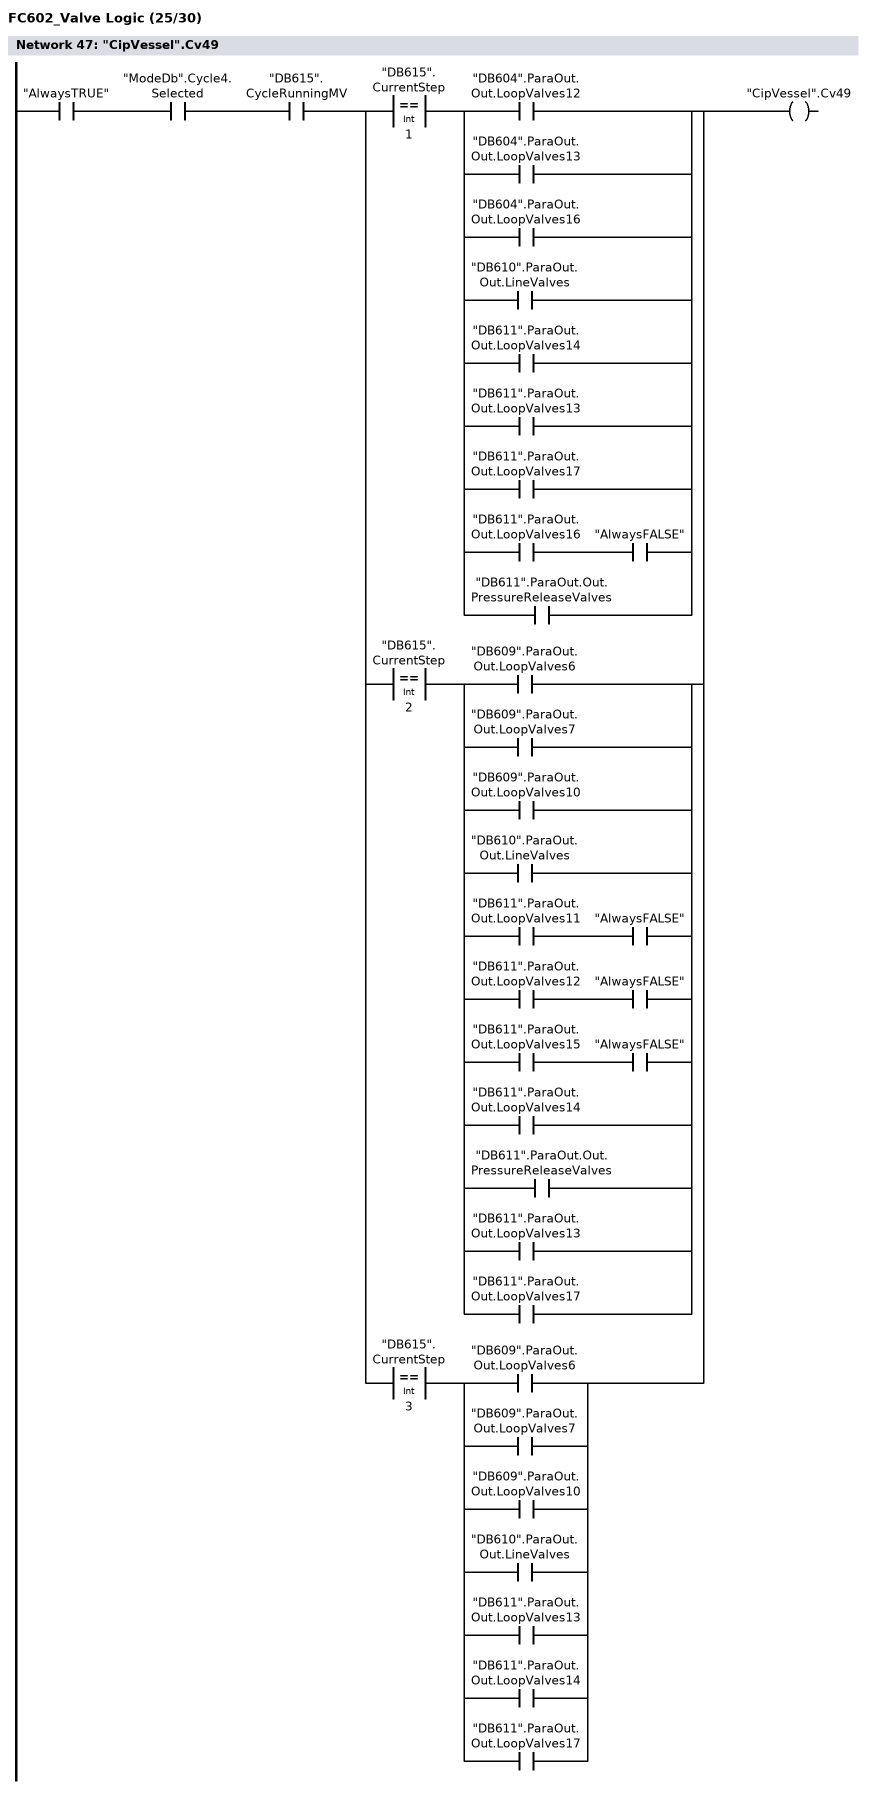
   RUNG wire#powerrail
      Contact( "AlwaysTRUE" )
      Contact( "ModeDb".Cycle4.Selected )
      Contact( "DB615".CycleRunningMV )
      wire#w1
      { S7_Templates := "SrcType := Int" } EQ_Contact(in1 := "DB615".CurrentStep, in2 := 1)
      wire#w2
      Contact( "DB604".ParaOut.Out.LoopValves12 )
      wire#w3
      Coil( "CipVessel".Cv49 )
   END_RUNG
   RUNG wire#w2
      Contact( "DB604".ParaOut.Out.LoopValves13 )
   END_RUNG wire#w3
   RUNG wire#w2
      Contact( "DB604".ParaOut.Out.LoopValves16 )
   END_RUNG wire#w3
   RUNG wire#w2
      Contact( "DB610".ParaOut.Out.LineValves )
   END_RUNG wire#w3
   RUNG wire#w2
      Contact( "DB611".ParaOut.Out.LoopValves14 )
   END_RUNG wire#w3
   RUNG wire#w2
      Contact( "DB611".ParaOut.Out.LoopValves13 )
   END_RUNG wire#w3
   RUNG wire#w2
      Contact( "DB611".ParaOut.Out.LoopValves17 )
   END_RUNG wire#w3
   RUNG wire#w2
      Contact( "DB611".ParaOut.Out.LoopValves16 )
      Contact( "AlwaysFALSE" )
   END_RUNG wire#w3
   RUNG wire#w2
      Contact( "DB611".ParaOut.Out.PressureReleaseValves )
   END_RUNG wire#w3
   RUNG wire#w1
      { S7_Templates := "SrcType := Int" } EQ_Contact(in1 := "DB615".CurrentStep, in2 := 2)
      wire#w4
      Contact( "DB609".ParaOut.Out.LoopValves6 )
   END_RUNG wire#w3
   RUNG wire#w4
      Contact( "DB609".ParaOut.Out.LoopValves7 )
   END_RUNG wire#w3
   RUNG wire#w4
      Contact( "DB609".ParaOut.Out.LoopValves10 )
   END_RUNG wire#w3
   RUNG wire#w4
      Contact( "DB610".ParaOut.Out.LineValves )
   END_RUNG wire#w3
   RUNG wire#w4
      Contact( "DB611".ParaOut.Out.LoopValves11 )
      Contact( "AlwaysFALSE" )
   END_RUNG wire#w3
   RUNG wire#w4
      Contact( "DB611".ParaOut.Out.LoopValves12 )
      Contact( "AlwaysFALSE" )
   END_RUNG wire#w3
   RUNG wire#w4
      Contact( "DB611".ParaOut.Out.LoopValves15 )
      Contact( "AlwaysFALSE" )
   END_RUNG wire#w3
   RUNG wire#w4
      Contact( "DB611".ParaOut.Out.LoopValves14 )
   END_RUNG wire#w3
   RUNG wire#w4
      Contact( "DB611".ParaOut.Out.PressureReleaseValves )
   END_RUNG wire#w3
   RUNG wire#w4
      Contact( "DB611".ParaOut.Out.LoopValves13 )
   END_RUNG wire#w3
   RUNG wire#w4
      Contact( "DB611".ParaOut.Out.LoopValves17 )
   END_RUNG wire#w3
   RUNG wire#w1
      { S7_Templates := "SrcType := Int" } EQ_Contact(in1 := "DB615".CurrentStep, in2 := 3)
      wire#w5
      Contact( "DB609".ParaOut.Out.LoopValves6 )
   END_RUNG wire#w3
   RUNG wire#w5
      Contact( "DB609".ParaOut.Out.LoopValves7 )
   END_RUNG wire#w3
   RUNG wire#w5
      Contact( "DB609".ParaOut.Out.LoopValves10 )
   END_RUNG wire#w3
   RUNG wire#w5
      Contact( "DB610".ParaOut.Out.LineValves )
   END_RUNG wire#w3
   RUNG wire#w5
      Contact( "DB611".ParaOut.Out.LoopValves13 )
   END_RUNG wire#w3
   RUNG wire#w5
      Contact( "DB611".ParaOut.Out.LoopValves14 )
   END_RUNG wire#w3
   RUNG wire#w5
      Contact( "DB611".ParaOut.Out.LoopValves17 )
   END_RUNG wire#w3
   // the same network as SCL:
   "CipVessel".Cv49 := "AlwaysTRUE" AND "ModeDb".Cycle4.Selected AND "DB615".CycleRunningMV AND ((("DB615".CurrentStep = 1) AND ("DB604".ParaOut.Out.LoopValves12 OR "DB604".ParaOut.Out.LoopValves13 OR "DB604".ParaOut.Out.LoopValves16 OR "DB610".ParaOut.Out.LineValves OR "DB611".ParaOut.Out.LoopValves14 OR "DB611".ParaOut.Out.LoopValves13 OR "DB611".ParaOut.Out.LoopValves17 OR ("DB611".ParaOut.Out.LoopValves16 AND "AlwaysFALSE") OR "DB611".ParaOut.Out.PressureReleaseValves)) OR (("DB615".CurrentStep = 2) AND ("DB609".ParaOut.Out.LoopValves6 OR "DB609".ParaOut.Out.LoopValves7 OR "DB609".ParaOut.Out.LoopValves10 OR "DB610".ParaOut.Out.LineValves OR ("DB611".ParaOut.Out.LoopValves11 AND "AlwaysFALSE") OR ("DB611".ParaOut.Out.LoopValves12 AND "AlwaysFALSE") OR ("DB611".ParaOut.Out.LoopValves15 AND "AlwaysFALSE") OR "DB611".ParaOut.Out.LoopValves14 OR "DB611".ParaOut.Out.PressureReleaseValves OR "DB611".ParaOut.Out.LoopValves13 OR "DB611".ParaOut.Out.LoopValves17)) OR (("DB615".CurrentStep = 3) AND ("DB609".ParaOut.Out.LoopValves6 OR "DB609".ParaOut.Out.LoopValves7 OR "DB609".ParaOut.Out.LoopValves10 OR "DB610".ParaOut.Out.LineValves OR "DB611".ParaOut.Out.LoopValves13 OR "DB611".ParaOut.Out.LoopValves14 OR "DB611".ParaOut.Out.LoopValves17)));
END_REGION

REGION Network 48: "CipVessel".Cv53
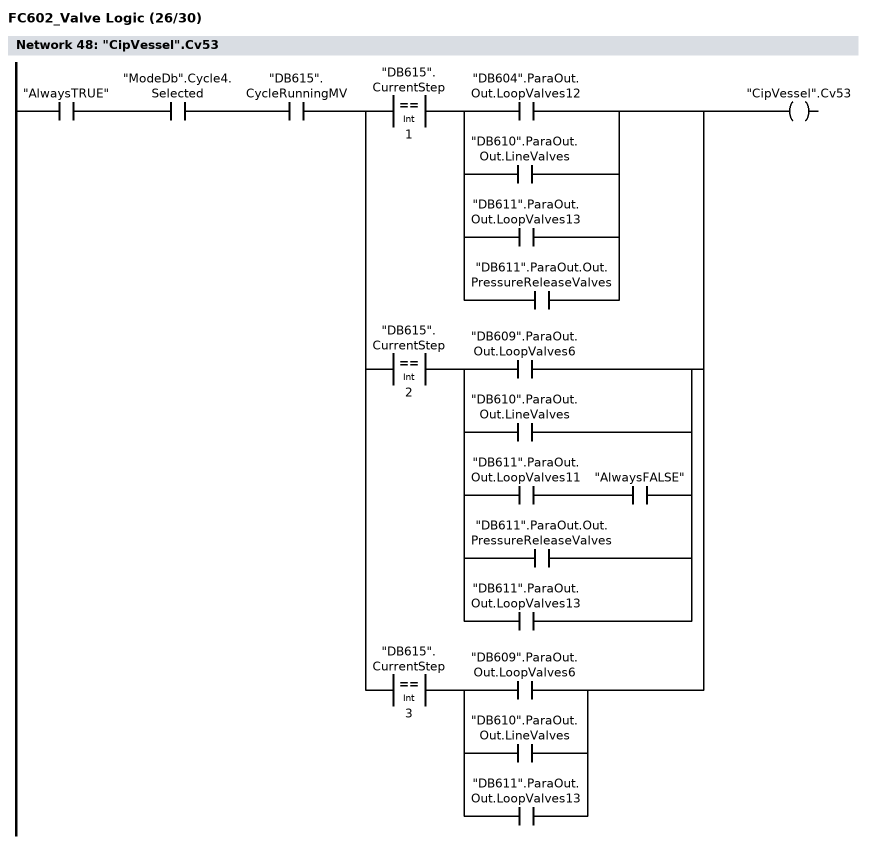
   RUNG wire#powerrail
      Contact( "AlwaysTRUE" )
      Contact( "ModeDb".Cycle4.Selected )
      Contact( "DB615".CycleRunningMV )
      wire#w1
      { S7_Templates := "SrcType := Int" } EQ_Contact(in1 := "DB615".CurrentStep, in2 := 1)
      wire#w2
      Contact( "DB604".ParaOut.Out.LoopValves12 )
      wire#w3
      Coil( "CipVessel".Cv53 )
   END_RUNG
   RUNG wire#w2
      Contact( "DB610".ParaOut.Out.LineValves )
   END_RUNG wire#w3
   RUNG wire#w2
      Contact( "DB611".ParaOut.Out.LoopValves13 )
   END_RUNG wire#w3
   RUNG wire#w2
      Contact( "DB611".ParaOut.Out.PressureReleaseValves )
   END_RUNG wire#w3
   RUNG wire#w1
      { S7_Templates := "SrcType := Int" } EQ_Contact(in1 := "DB615".CurrentStep, in2 := 2)
      wire#w4
      Contact( "DB609".ParaOut.Out.LoopValves6 )
   END_RUNG wire#w3
   RUNG wire#w4
      Contact( "DB610".ParaOut.Out.LineValves )
   END_RUNG wire#w3
   RUNG wire#w4
      Contact( "DB611".ParaOut.Out.LoopValves11 )
      Contact( "AlwaysFALSE" )
   END_RUNG wire#w3
   RUNG wire#w4
      Contact( "DB611".ParaOut.Out.PressureReleaseValves )
   END_RUNG wire#w3
   RUNG wire#w4
      Contact( "DB611".ParaOut.Out.LoopValves13 )
   END_RUNG wire#w3
   RUNG wire#w1
      { S7_Templates := "SrcType := Int" } EQ_Contact(in1 := "DB615".CurrentStep, in2 := 3)
      wire#w5
      Contact( "DB609".ParaOut.Out.LoopValves6 )
   END_RUNG wire#w3
   RUNG wire#w5
      Contact( "DB610".ParaOut.Out.LineValves )
   END_RUNG wire#w3
   RUNG wire#w5
      Contact( "DB611".ParaOut.Out.LoopValves13 )
   END_RUNG wire#w3
   // the same network as SCL:
   "CipVessel".Cv53 := "AlwaysTRUE" AND "ModeDb".Cycle4.Selected AND "DB615".CycleRunningMV AND ((("DB615".CurrentStep = 1) AND ("DB604".ParaOut.Out.LoopValves12 OR "DB610".ParaOut.Out.LineValves OR "DB611".ParaOut.Out.LoopValves13 OR "DB611".ParaOut.Out.PressureReleaseValves)) OR (("DB615".CurrentStep = 2) AND ("DB609".ParaOut.Out.LoopValves6 OR "DB610".ParaOut.Out.LineValves OR ("DB611".ParaOut.Out.LoopValves11 AND "AlwaysFALSE") OR "DB611".ParaOut.Out.PressureReleaseValves OR "DB611".ParaOut.Out.LoopValves13)) OR (("DB615".CurrentStep = 3) AND ("DB609".ParaOut.Out.LoopValves6 OR "DB610".ParaOut.Out.LineValves OR "DB611".ParaOut.Out.LoopValves13)));
END_REGION

REGION Network 49: ----------- PF02 OUT -------------
END_REGION

REGION Network 50: "CipVessel".Cv56
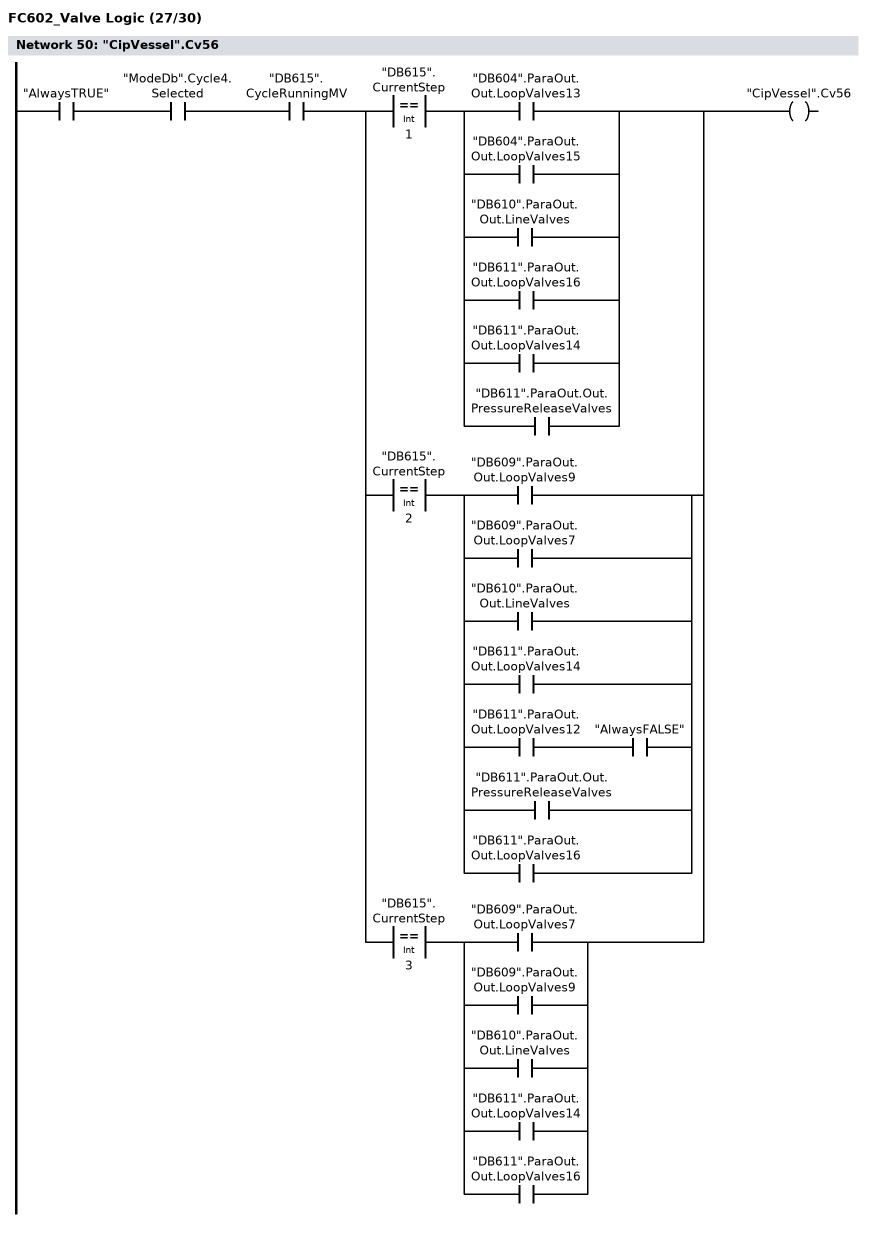
   RUNG wire#powerrail
      Contact( "AlwaysTRUE" )
      Contact( "ModeDb".Cycle4.Selected )
      Contact( "DB615".CycleRunningMV )
      wire#w1
      { S7_Templates := "SrcType := Int" } EQ_Contact(in1 := "DB615".CurrentStep, in2 := 1)
      wire#w2
      Contact( "DB604".ParaOut.Out.LoopValves13 )
      wire#w3
      Coil( "CipVessel".Cv56 )
   END_RUNG
   RUNG wire#w2
      Contact( "DB604".ParaOut.Out.LoopValves15 )
   END_RUNG wire#w3
   RUNG wire#w2
      Contact( "DB610".ParaOut.Out.LineValves )
   END_RUNG wire#w3
   RUNG wire#w2
      Contact( "DB611".ParaOut.Out.LoopValves16 )
   END_RUNG wire#w3
   RUNG wire#w2
      Contact( "DB611".ParaOut.Out.LoopValves14 )
   END_RUNG wire#w3
   RUNG wire#w2
      Contact( "DB611".ParaOut.Out.PressureReleaseValves )
   END_RUNG wire#w3
   RUNG wire#w1
      { S7_Templates := "SrcType := Int" } EQ_Contact(in1 := "DB615".CurrentStep, in2 := 2)
      wire#w4
      Contact( "DB609".ParaOut.Out.LoopValves9 )
   END_RUNG wire#w3
   RUNG wire#w4
      Contact( "DB609".ParaOut.Out.LoopValves7 )
   END_RUNG wire#w3
   RUNG wire#w4
      Contact( "DB610".ParaOut.Out.LineValves )
   END_RUNG wire#w3
   RUNG wire#w4
      Contact( "DB611".ParaOut.Out.LoopValves14 )
   END_RUNG wire#w3
   RUNG wire#w4
      Contact( "DB611".ParaOut.Out.LoopValves12 )
      Contact( "AlwaysFALSE" )
   END_RUNG wire#w3
   RUNG wire#w4
      Contact( "DB611".ParaOut.Out.PressureReleaseValves )
   END_RUNG wire#w3
   RUNG wire#w4
      Contact( "DB611".ParaOut.Out.LoopValves16 )
   END_RUNG wire#w3
   RUNG wire#w1
      { S7_Templates := "SrcType := Int" } EQ_Contact(in1 := "DB615".CurrentStep, in2 := 3)
      wire#w5
      Contact( "DB609".ParaOut.Out.LoopValves7 )
   END_RUNG wire#w3
   RUNG wire#w5
      Contact( "DB609".ParaOut.Out.LoopValves9 )
   END_RUNG wire#w3
   RUNG wire#w5
      Contact( "DB610".ParaOut.Out.LineValves )
   END_RUNG wire#w3
   RUNG wire#w5
      Contact( "DB611".ParaOut.Out.LoopValves14 )
   END_RUNG wire#w3
   RUNG wire#w5
      Contact( "DB611".ParaOut.Out.LoopValves16 )
   END_RUNG wire#w3
   // the same network as SCL:
   "CipVessel".Cv56 := "AlwaysTRUE" AND "ModeDb".Cycle4.Selected AND "DB615".CycleRunningMV AND ((("DB615".CurrentStep = 1) AND ("DB604".ParaOut.Out.LoopValves13 OR "DB604".ParaOut.Out.LoopValves15 OR "DB610".ParaOut.Out.LineValves OR "DB611".ParaOut.Out.LoopValves16 OR "DB611".ParaOut.Out.LoopValves14 OR "DB611".ParaOut.Out.PressureReleaseValves)) OR (("DB615".CurrentStep = 2) AND ("DB609".ParaOut.Out.LoopValves9 OR "DB609".ParaOut.Out.LoopValves7 OR "DB610".ParaOut.Out.LineValves OR "DB611".ParaOut.Out.LoopValves14 OR ("DB611".ParaOut.Out.LoopValves12 AND "AlwaysFALSE") OR "DB611".ParaOut.Out.PressureReleaseValves OR "DB611".ParaOut.Out.LoopValves16)) OR (("DB615".CurrentStep = 3) AND ("DB609".ParaOut.Out.LoopValves7 OR "DB609".ParaOut.Out.LoopValves9 OR "DB610".ParaOut.Out.LineValves OR "DB611".ParaOut.Out.LoopValves14 OR "DB611".ParaOut.Out.LoopValves16)));
END_REGION

REGION Network 51: "CipVessel".Cv57
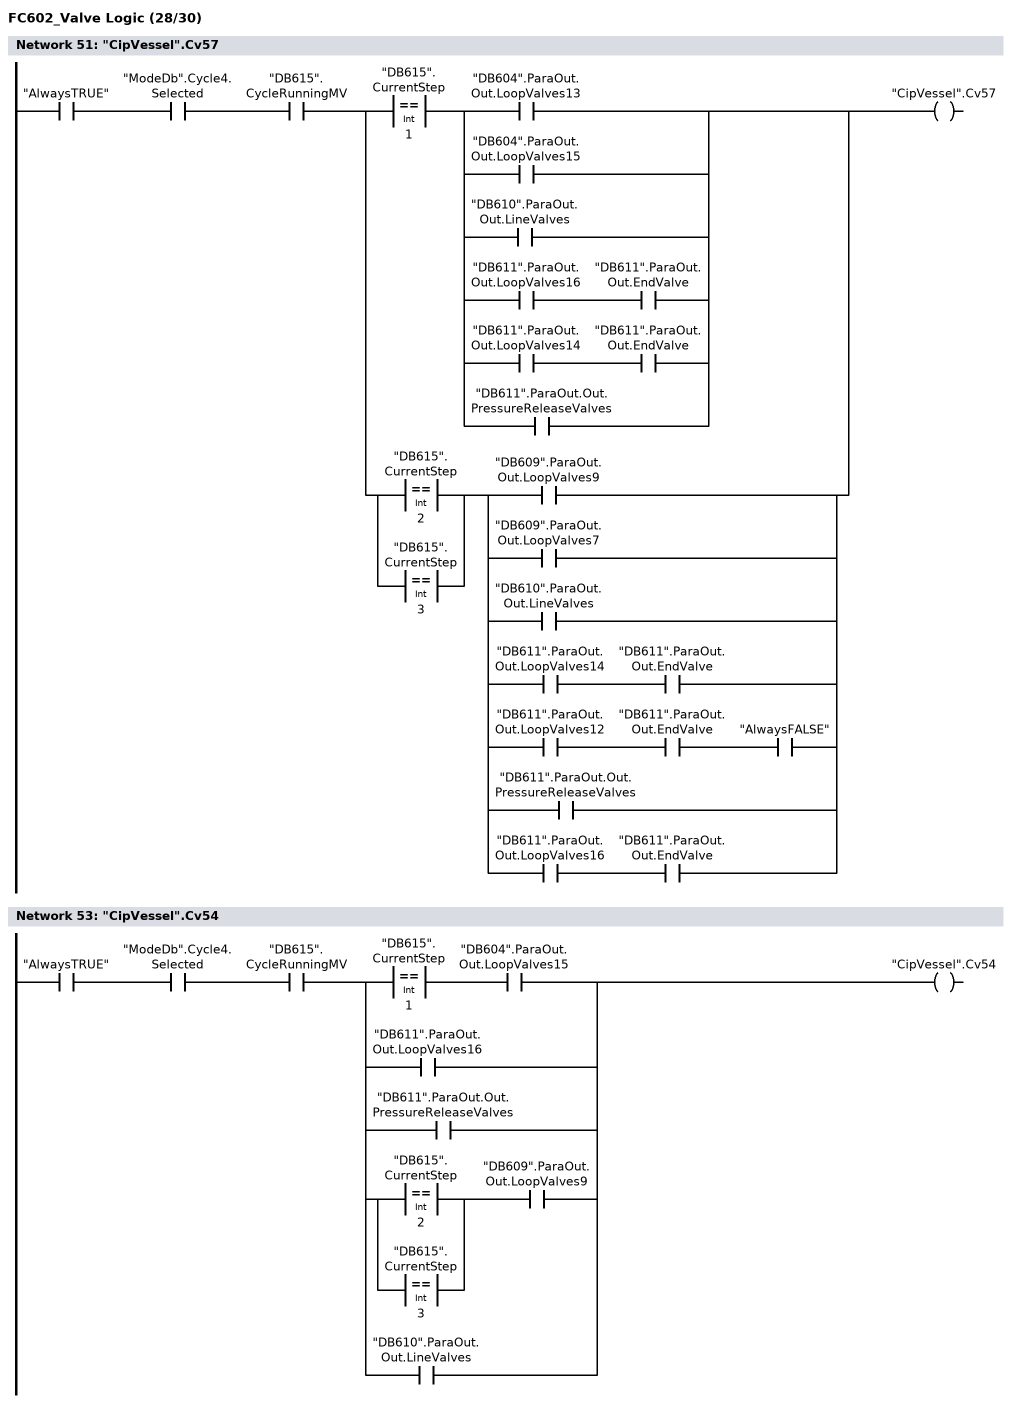
   RUNG wire#powerrail
      Contact( "AlwaysTRUE" )
      Contact( "ModeDb".Cycle4.Selected )
      Contact( "DB615".CycleRunningMV )
      wire#w1
      { S7_Templates := "SrcType := Int" } EQ_Contact(in1 := "DB615".CurrentStep, in2 := 1)
      wire#w2
      Contact( "DB604".ParaOut.Out.LoopValves13 )
      wire#w3
      Coil( "CipVessel".Cv57 )
   END_RUNG
   RUNG wire#w2
      Contact( "DB604".ParaOut.Out.LoopValves15 )
   END_RUNG wire#w3
   RUNG wire#w2
      Contact( "DB610".ParaOut.Out.LineValves )
   END_RUNG wire#w3
   RUNG wire#w2
      Contact( "DB611".ParaOut.Out.LoopValves16 )
      Contact( "DB611".ParaOut.Out.EndValve )
   END_RUNG wire#w3
   RUNG wire#w2
      Contact( "DB611".ParaOut.Out.LoopValves14 )
      Contact( "DB611".ParaOut.Out.EndValve )
   END_RUNG wire#w3
   RUNG wire#w2
      Contact( "DB611".ParaOut.Out.PressureReleaseValves )
   END_RUNG wire#w3
   RUNG wire#w1
      { S7_Templates := "SrcType := Int" } EQ_Contact(in1 := "DB615".CurrentStep, in2 := 2)
      wire#w4
      Contact( "DB609".ParaOut.Out.LoopValves9 )
   END_RUNG wire#w3
   RUNG wire#w1
      { S7_Templates := "SrcType := Int" } EQ_Contact(in1 := "DB615".CurrentStep, in2 := 3)
   END_RUNG wire#w4
   RUNG wire#w4
      Contact( "DB609".ParaOut.Out.LoopValves7 )
   END_RUNG wire#w3
   RUNG wire#w4
      Contact( "DB610".ParaOut.Out.LineValves )
   END_RUNG wire#w3
   RUNG wire#w4
      Contact( "DB611".ParaOut.Out.LoopValves14 )
      Contact( "DB611".ParaOut.Out.EndValve )
   END_RUNG wire#w3
   RUNG wire#w4
      Contact( "DB611".ParaOut.Out.LoopValves12 )
      Contact( "DB611".ParaOut.Out.EndValve )
      Contact( "AlwaysFALSE" )
   END_RUNG wire#w3
   RUNG wire#w4
      Contact( "DB611".ParaOut.Out.PressureReleaseValves )
   END_RUNG wire#w3
   RUNG wire#w4
      Contact( "DB611".ParaOut.Out.LoopValves16 )
      Contact( "DB611".ParaOut.Out.EndValve )
   END_RUNG wire#w3
   // the same network as SCL:
   "CipVessel".Cv57 := "AlwaysTRUE" AND "ModeDb".Cycle4.Selected AND "DB615".CycleRunningMV AND ((("DB615".CurrentStep = 1) AND ("DB604".ParaOut.Out.LoopValves13 OR "DB604".ParaOut.Out.LoopValves15 OR "DB610".ParaOut.Out.LineValves OR ("DB611".ParaOut.Out.LoopValves16 AND "DB611".ParaOut.Out.EndValve) OR ("DB611".ParaOut.Out.LoopValves14 AND "DB611".ParaOut.Out.EndValve) OR "DB611".ParaOut.Out.PressureReleaseValves)) OR ((("DB615".CurrentStep = 2) OR ("DB615".CurrentStep = 3)) AND ("DB609".ParaOut.Out.LoopValves9 OR "DB609".ParaOut.Out.LoopValves7 OR "DB610".ParaOut.Out.LineValves OR ("DB611".ParaOut.Out.LoopValves14 AND "DB611".ParaOut.Out.EndValve) OR ("DB611".ParaOut.Out.LoopValves12 AND "DB611".ParaOut.Out.EndValve AND "AlwaysFALSE") OR "DB611".ParaOut.Out.PressureReleaseValves OR ("DB611".ParaOut.Out.LoopValves16 AND "DB611".ParaOut.Out.EndValve))));
END_REGION

REGION Network 52: ---------- PTL LINE ------------
END_REGION

REGION Network 53: "CipVessel".Cv54
   RUNG wire#powerrail
      Contact( "AlwaysTRUE" )
      Contact( "ModeDb".Cycle4.Selected )
      Contact( "DB615".CycleRunningMV )
      wire#w1
      { S7_Templates := "SrcType := Int" } EQ_Contact(in1 := "DB615".CurrentStep, in2 := 1)
      Contact( "DB604".ParaOut.Out.LoopValves15 )
      wire#w2
      Coil( "CipVessel".Cv54 )
   END_RUNG
   RUNG wire#w1
      Contact( "DB611".ParaOut.Out.LoopValves16 )
   END_RUNG wire#w2
   RUNG wire#w1
      Contact( "DB611".ParaOut.Out.PressureReleaseValves )
   END_RUNG wire#w2
   RUNG wire#w1
      { S7_Templates := "SrcType := Int" } EQ_Contact(in1 := "DB615".CurrentStep, in2 := 2)
      wire#w3
      Contact( "DB609".ParaOut.Out.LoopValves9 )
   END_RUNG wire#w2
   RUNG wire#w1
      { S7_Templates := "SrcType := Int" } EQ_Contact(in1 := "DB615".CurrentStep, in2 := 3)
   END_RUNG wire#w3
   RUNG wire#w1
      Contact( "DB610".ParaOut.Out.LineValves )
   END_RUNG wire#w2
   // the same network as SCL:
   "CipVessel".Cv54 := "AlwaysTRUE" AND "ModeDb".Cycle4.Selected AND "DB615".CycleRunningMV AND ((("DB615".CurrentStep = 1) AND "DB604".ParaOut.Out.LoopValves15) OR "DB611".ParaOut.Out.LoopValves16 OR "DB611".ParaOut.Out.PressureReleaseValves OR ((("DB615".CurrentStep = 2) OR ("DB615".CurrentStep = 3)) AND "DB609".ParaOut.Out.LoopValves9) OR "DB610".ParaOut.Out.LineValves);
END_REGION

REGION Network 54: "CipVessel".Cv55
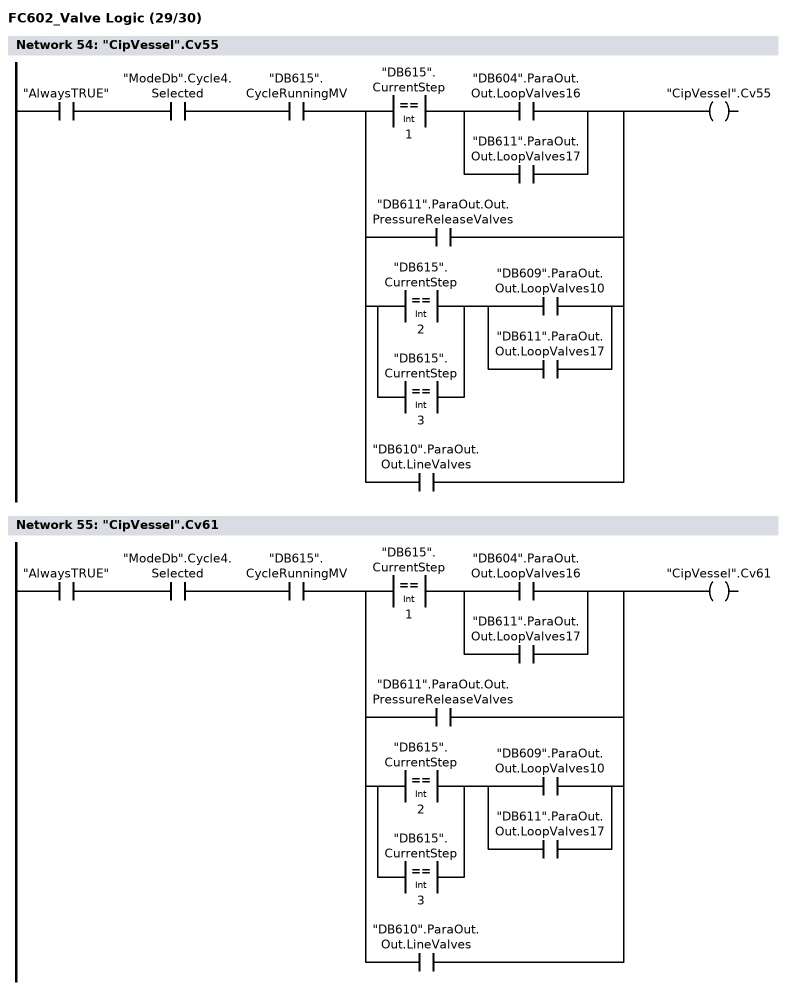
   RUNG wire#powerrail
      Contact( "AlwaysTRUE" )
      Contact( "ModeDb".Cycle4.Selected )
      Contact( "DB615".CycleRunningMV )
      wire#w1
      { S7_Templates := "SrcType := Int" } EQ_Contact(in1 := "DB615".CurrentStep, in2 := 1)
      wire#w2
      Contact( "DB604".ParaOut.Out.LoopValves16 )
      wire#w3
      Coil( "CipVessel".Cv55 )
   END_RUNG
   RUNG wire#w2
      Contact( "DB611".ParaOut.Out.LoopValves17 )
   END_RUNG wire#w3
   RUNG wire#w1
      Contact( "DB611".ParaOut.Out.PressureReleaseValves )
   END_RUNG wire#w3
   RUNG wire#w1
      { S7_Templates := "SrcType := Int" } EQ_Contact(in1 := "DB615".CurrentStep, in2 := 2)
      wire#w4
      Contact( "DB609".ParaOut.Out.LoopValves10 )
   END_RUNG wire#w3
   RUNG wire#w1
      { S7_Templates := "SrcType := Int" } EQ_Contact(in1 := "DB615".CurrentStep, in2 := 3)
   END_RUNG wire#w4
   RUNG wire#w4
      Contact( "DB611".ParaOut.Out.LoopValves17 )
   END_RUNG wire#w3
   RUNG wire#w1
      Contact( "DB610".ParaOut.Out.LineValves )
   END_RUNG wire#w3
   // the same network as SCL:
   "CipVessel".Cv55 := "AlwaysTRUE" AND "ModeDb".Cycle4.Selected AND "DB615".CycleRunningMV AND ((("DB615".CurrentStep = 1) AND ("DB604".ParaOut.Out.LoopValves16 OR "DB611".ParaOut.Out.LoopValves17)) OR "DB611".ParaOut.Out.PressureReleaseValves OR ((("DB615".CurrentStep = 2) OR ("DB615".CurrentStep = 3)) AND ("DB609".ParaOut.Out.LoopValves10 OR "DB611".ParaOut.Out.LoopValves17)) OR "DB610".ParaOut.Out.LineValves);
END_REGION

REGION Network 55: "CipVessel".Cv61
   RUNG wire#powerrail
      Contact( "AlwaysTRUE" )
      Contact( "ModeDb".Cycle4.Selected )
      Contact( "DB615".CycleRunningMV )
      wire#w1
      { S7_Templates := "SrcType := Int" } EQ_Contact(in1 := "DB615".CurrentStep, in2 := 1)
      wire#w2
      Contact( "DB604".ParaOut.Out.LoopValves16 )
      wire#w3
      Coil( "CipVessel".Cv61 )
   END_RUNG
   RUNG wire#w2
      Contact( "DB611".ParaOut.Out.LoopValves17 )
   END_RUNG wire#w3
   RUNG wire#w1
      Contact( "DB611".ParaOut.Out.PressureReleaseValves )
   END_RUNG wire#w3
   RUNG wire#w1
      { S7_Templates := "SrcType := Int" } EQ_Contact(in1 := "DB615".CurrentStep, in2 := 2)
      wire#w4
      Contact( "DB609".ParaOut.Out.LoopValves10 )
   END_RUNG wire#w3
   RUNG wire#w1
      { S7_Templates := "SrcType := Int" } EQ_Contact(in1 := "DB615".CurrentStep, in2 := 3)
   END_RUNG wire#w4
   RUNG wire#w4
      Contact( "DB611".ParaOut.Out.LoopValves17 )
   END_RUNG wire#w3
   RUNG wire#w1
      Contact( "DB610".ParaOut.Out.LineValves )
   END_RUNG wire#w3
   // the same network as SCL:
   "CipVessel".Cv61 := "AlwaysTRUE" AND "ModeDb".Cycle4.Selected AND "DB615".CycleRunningMV AND ((("DB615".CurrentStep = 1) AND ("DB604".ParaOut.Out.LoopValves16 OR "DB611".ParaOut.Out.LoopValves17)) OR "DB611".ParaOut.Out.PressureReleaseValves OR ((("DB615".CurrentStep = 2) OR ("DB615".CurrentStep = 3)) AND ("DB609".ParaOut.Out.LoopValves10 OR "DB611".ParaOut.Out.LoopValves17)) OR "DB610".ParaOut.Out.LineValves);
END_REGION

REGION Network 56: "CipVessel".Cv60
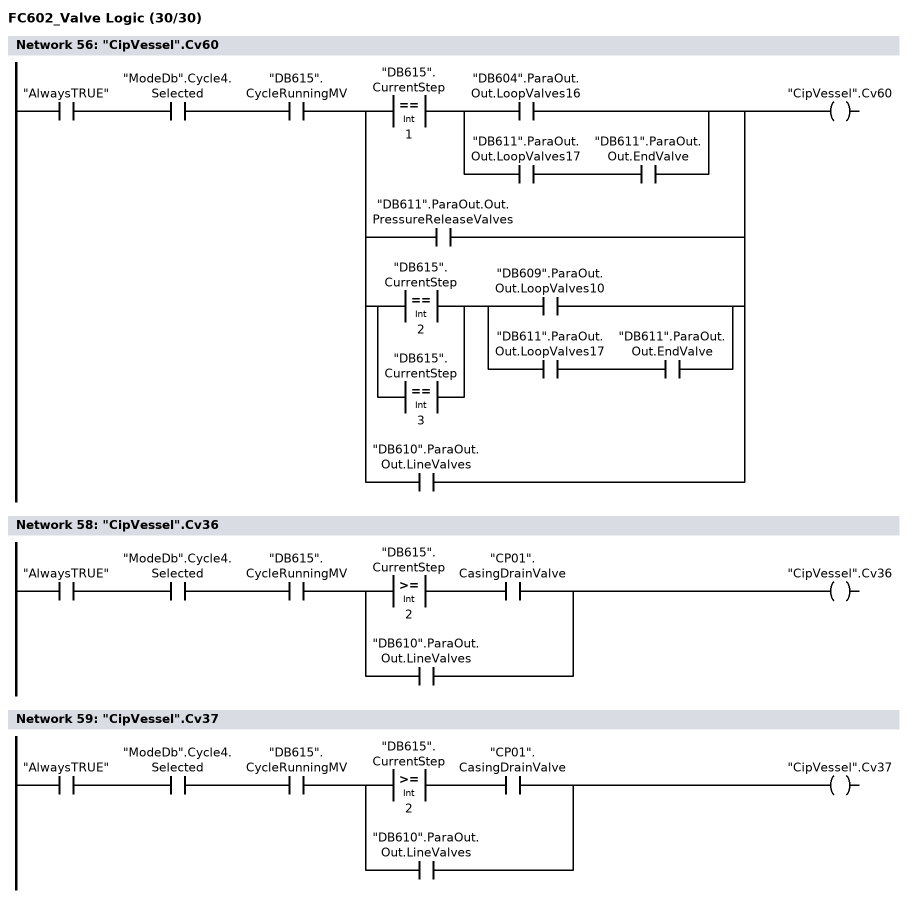
   RUNG wire#powerrail
      Contact( "AlwaysTRUE" )
      Contact( "ModeDb".Cycle4.Selected )
      Contact( "DB615".CycleRunningMV )
      wire#w1
      { S7_Templates := "SrcType := Int" } EQ_Contact(in1 := "DB615".CurrentStep, in2 := 1)
      wire#w2
      Contact( "DB604".ParaOut.Out.LoopValves16 )
      wire#w3
      Coil( "CipVessel".Cv60 )
   END_RUNG
   RUNG wire#w2
      Contact( "DB611".ParaOut.Out.LoopValves17 )
      Contact( "DB611".ParaOut.Out.EndValve )
   END_RUNG wire#w3
   RUNG wire#w1
      Contact( "DB611".ParaOut.Out.PressureReleaseValves )
   END_RUNG wire#w3
   RUNG wire#w1
      { S7_Templates := "SrcType := Int" } EQ_Contact(in1 := "DB615".CurrentStep, in2 := 2)
      wire#w4
      Contact( "DB609".ParaOut.Out.LoopValves10 )
   END_RUNG wire#w3
   RUNG wire#w1
      { S7_Templates := "SrcType := Int" } EQ_Contact(in1 := "DB615".CurrentStep, in2 := 3)
   END_RUNG wire#w4
   RUNG wire#w4
      Contact( "DB611".ParaOut.Out.LoopValves17 )
      Contact( "DB611".ParaOut.Out.EndValve )
   END_RUNG wire#w3
   RUNG wire#w1
      Contact( "DB610".ParaOut.Out.LineValves )
   END_RUNG wire#w3
   // the same network as SCL:
   "CipVessel".Cv60 := "AlwaysTRUE" AND "ModeDb".Cycle4.Selected AND "DB615".CycleRunningMV AND ((("DB615".CurrentStep = 1) AND ("DB604".ParaOut.Out.LoopValves16 OR ("DB611".ParaOut.Out.LoopValves17 AND "DB611".ParaOut.Out.EndValve))) OR "DB611".ParaOut.Out.PressureReleaseValves OR ((("DB615".CurrentStep = 2) OR ("DB615".CurrentStep = 3)) AND ("DB609".ParaOut.Out.LoopValves10 OR ("DB611".ParaOut.Out.LoopValves17 AND "DB611".ParaOut.Out.EndValve))) OR "DB610".ParaOut.Out.LineValves);
END_REGION

REGION Network 57: ----------PCD DRAIN------------
END_REGION

REGION Network 58: "CipVessel".Cv36
   RUNG wire#powerrail
      Contact( "AlwaysTRUE" )
      Contact( "ModeDb".Cycle4.Selected )
      Contact( "DB615".CycleRunningMV )
      wire#w1
      { S7_Templates := "SrcType := Int" } GE_Contact(in1 := "DB615".CurrentStep, in2 := 2)
      Contact( "CP01".CasingDrainValve )
      wire#w2
      Coil( "CipVessel".Cv36 )
   END_RUNG
   RUNG wire#w1
      Contact( "DB610".ParaOut.Out.LineValves )
   END_RUNG wire#w2
   // the same network as SCL:
   "CipVessel".Cv36 := "AlwaysTRUE" AND "ModeDb".Cycle4.Selected AND "DB615".CycleRunningMV AND ((("DB615".CurrentStep >= 2) AND "CP01".CasingDrainValve) OR "DB610".ParaOut.Out.LineValves);
END_REGION

REGION Network 59: "CipVessel".Cv37
   RUNG wire#powerrail
      Contact( "AlwaysTRUE" )
      Contact( "ModeDb".Cycle4.Selected )
      Contact( "DB615".CycleRunningMV )
      wire#w1
      { S7_Templates := "SrcType := Int" } GE_Contact(in1 := "DB615".CurrentStep, in2 := 2)
      Contact( "CP01".CasingDrainValve )
      wire#w2
      Coil( "CipVessel".Cv37 )
   END_RUNG
   RUNG wire#w1
      Contact( "DB610".ParaOut.Out.LineValves )
   END_RUNG wire#w2
   // the same network as SCL:
   "CipVessel".Cv37 := "AlwaysTRUE" AND "ModeDb".Cycle4.Selected AND "DB615".CycleRunningMV AND ((("DB615".CurrentStep >= 2) AND "CP01".CasingDrainValve) OR "DB610".ParaOut.Out.LineValves);
END_REGION
END_FUNCTION
